PROGRAM MAIN_Orden_Lectura_PLCs
VAR
	bHabilitarLecturaDePLCs : BOOL := TRUE;
	bHabilitaLectura_Maestro : BOOL:=TRUE;
	State_Lectura_PLC: (READING_PLC_WAITING, READING_PLC_MAESTRO, FINISH_ALL_OK);
	tReadState_Entre_Lecturas_PLCs:ton:=(PT:=T#5MS);
END_VAR

// POU para ordenar la lectura de los distintos PLCs para que nunca lean a la vez 

CASE State_Lectura_PLC OF 

	READING_PLC_WAITING:tReadState_Entre_Lecturas_PLCs(IN:=FALSE);	

	READING_PLC_MAESTRO:	IF bHabilitaLectura_Maestro THEN
						tReadState_Entre_Lecturas_PLCs(IN:=TRUE);	
							IF tReadState_Entre_Lecturas_PLCs.Q THEN 
								tReadState_Entre_Lecturas_PLCs(IN:=FALSE);
								Lectura_Maestro();
								Lectura_Maestro.fbLectura_a_PLC_Maestro.SetStartReading();
							END_IF
							IF Lectura_Maestro.bNextBlockToRead_L4_Done THEN

								Lectura_Maestro.fbLectura_a_PLC_Maestro.SetFalseBlockReadDone();
								State_Lectura_PLC := FINISH_ALL_OK; //Cuando se añada un PLC cambiad el nombre.
							END_IF
						ELSE 
							State_Lectura_PLC := FINISH_ALL_OK; //Cuando se añada un PLC cambiad el nombre.
							Lectura_Maestro.fbLectura_a_PLC_Maestro.SetFalseBlockReadDone();
					END_IF
					
	FINISH_ALL_OK: tReadState_Entre_Lecturas_PLCs(IN:=FALSE);	
					State_Lectura_PLC := READING_PLC_Maestro;				

END_CASE



//Habilitar la lectura de los PLCs
IF bHabilitarLecturaDePLCs THEN 
	SetStartReadingPLCs();
	ELSE
		State_Lectura_PLC:=READING_PLC_WAITING;
END_IF

METHOD SetStartReadingPLCs : BOOL
VAR_INPUT
END_VAR
IF State_Lectura_PLC = READING_PLC_WAITING THEN 
	State_Lectura_PLC := READING_PLC_Maestro;
END_IF
END_METHOD

END_PROGRAM

(* stored: Version 1.1.0.1, ProductVersion 3.1.4024.12
   POU MAIN_Orden_Lectura_PLCs: Id {2ed88424-2e1b-40b4-a24d-83029be2134a}, SpecialFunc None
   Method SetStartReadingPLCs: Id {194546da-c227-4ee3-b58c-ae619e79be05} *)
